Fanuc TP program (LS listing): _clamp_out.ls

/PROG  _CLAMP_OUT
/ATTR
OWNER		= MNEDITOR;
COMMENT		= "";
PROG_SIZE	= 229;
CREATE		= DATE 26-06-12  TIME 05:50:48;
MODIFIED	= DATE 26-06-12  TIME 05:51:08;
FILE_NAME	= _CLAMP_I;
VERSION		= 0;
LINE_COUNT	= 2;
MEMORY_SIZE	= 593;
PROTECT		= READ_WRITE;
TCD:  STACK_SIZE	= 0,
      TASK_PRIORITY	= 50,
      TIME_SLICE	= 0,
      BUSY_LAMP_OFF	= 0,
      ABORT_REQUEST	= 0,
      PAUSE_REQUEST	= 0;
DEFAULT_GROUP	= 1,*,*,*,*;
CONTROL_CODE	= 00000000 00000000;
LOCAL_REGISTERS	= 0,0,0;
/APPL

AUTO_SINGULARITY_HEADER;
  ENABLE_SINGULARITY_AVOIDANCE   : TRUE;
/MN
   1:  DO[68:OFF:Ret Hook-Open]=ON ;
   2:  DO[67:OFF:Ext Hook-Closed]=OFF ;
/POS
/END
